KUKA KRL program: main.src, main.dat

--- main.src ---
&ACCESS RVP
&REL 135
&PARAM EDITMASK = *
&PARAM TEMPLATE = C:\KRC\Roboter\Template\vorgabe
&PARAM DISKPATH = KRC:\R1\Program
DEF main( )
;fold FRAME
DECL FRAME READY_POS
DECL FRAME stack_POS
DECL FRAME up_pos
DECL FRAME stack_end
DECL FRAME rotation_pos
DECL INT X
;endfold
;FOLD INI;%{PE}
  ;FOLD BASISTECH INI
    GLOBAL INTERRUPT DECL 3 WHEN $STOPMESS==TRUE DO IR_STOPM ( )
    INTERRUPT ON 3
    BAS (#INITMOV,0 )
  ;ENDFOLD (BASISTECH INI)
  ;FOLD USER INI
    ;Make your modifications here

  ;ENDFOLD (USER INI)
;ENDFOLD (INI)
;FOLD PTP HOME  Vel= 100 % DEFAULT;%{PE}%MKUKATPBASIS,%CMOVE,%VPTP,%P 1:PTP, 2:HOME, 3:, 5:100, 7:DEFAULT
$BWDSTART = FALSE
PDAT_ACT=PDEFAULT
FDAT_ACT=FHOME
BAS (#PTP_PARAMS,100 )
$H_POS=XHOME
PTP  XHOME
;ENDFOLD
if false then
;FOLD PTP maduo Vel=100 % PDAT1 Tool[1]:test Base[1]:tesy;%{PE}%R 8.3.44,%MKUKATPBASIS,%CMOVE,%VPTP,%P 1:PTP, 2:maduo, 3:, 5:100, 7:PDAT1
$BWDSTART=FALSE
PDAT_ACT=PPDAT1
FDAT_ACT=Fmaduo
BAS(#PTP_PARAMS,100)
PTP Xmaduo
;ENDFOLD
endif
loop
continue
$advance=3
;FOLD USER INI
$out[2]=FALSE
$OUT[3]=false
$OUT[4]=false
;ENDFOLD
$advance=3
;PTP Pick_Up
;FOLD PTP pick_up CONT Vel=100 % PDAT3 Tool[1]:test Base[1]:tesy;%{PE}%R 8.3.44,%MKUKATPBASIS,%CMOVE,%VPTP,%P 1:PTP, 2:pick_up, 3:C_DIS, 5:100, 7:PDAT3
$BWDSTART=FALSE
PDAT_ACT=PPDAT3
FDAT_ACT=Fpick_up
BAS(#PTP_PARAMS,100)
PTP Xpick_up C_DIS
;ENDFOLD
continue
;wait for $in[1] and $in[2] AND $aut ;wait allow Pick
wait sec 0
$ov_pro=100
$advance=3
;PTP pick_Up
$out[3]=true
calculation()
CONTINUE
;start rotation
;START TO MADUO
;START
;fold READY_POS
READY_POS=Xmaduo
ready_POS.X=ready_pos.X+P_POSITION[num,tier].X
ready_pos.y=ready_pos.y+P_POSITION[num,tier].y
READY_POS.Z=READY_POS.Z+RH
$BASE=BASE_DATA[1]
FOR X=1 TO 6
$VEL_AXIS[X]=85
$ACC_AXIS[X]=85
ENDFOR
$APO.CPTP=5
ptp READY_POS C_DIS
;endfold
; stack start
;FOLD STACK_POS
stack_POS=Xmaduo
stack_POS.X=stack_POS.X+P_POSITION[num,tier].X
stack_POS.y=stack_POS.y+P_POSITION[num,tier].y
$BASE=BASE_DATA[1]
FOR X=1 TO 6
$VEL_AXIS[X]=85
$ACC_AXIS[X]=85
ENDFOR
$APO.CPTP=5
ptp stack_POS C_DIS
;ENDFOLD
$OUT[2]=FALSE
$OUT[4]=true
wait sec 1
;fold READY_POS
READY_POS=Xmaduo
ready_pos.X=ready_pos.X+P_POSITION[num,tier].X
ready_pos.y=ready_pos.y+P_POSITION[num,tier].y
READY_POS.Z=READY_POS.Z+RH
$BASE=BASE_DATA[1]
FOR X=1 TO 6
$VEL_AXIS[X]=85
$ACC_AXIS[X]=85
ENDFOR
$APO.CPTP=5
ptp READY_POS C_DIS
;endfold
$advance=3
;STACK END
$out[3]=false
$out[4]=false
$ov_pro=100
;FOLD COUNT
Tier=Tier+1
if Tier>3 then
   NUM=Num+1
tier=1

endif
if num>4 then
num=1
exit
endif

;ENDFOLD
endloop
;FOLD PTP HOME Vel=100 % DEFAULT;%{PE}%R 8.3.44,%MKUKATPBASIS,%CMOVE,%VPTP,%P 1:PTP, 2:HOME, 3:, 5:100, 7:DEFAULT
$BWDSTART=FALSE
PDAT_ACT=PDEFAULT
FDAT_ACT=FHOME
BAS(#PTP_PARAMS,100)
$H_POS=XHOME
PTP XHOME
;ENDFOLD
END

--- main.dat ---
&ACCESS RVP
&REL 135
&PARAM EDITMASK = *
&PARAM TEMPLATE = C:\KRC\Roboter\Template\vorgabe
&PARAM DISKPATH = KRC:\R1\Program
DEFDAT  main
;FOLD EXTERNAL DECLARATIONS;%{PE}%MKUKATPBASIS,%CEXT,%VCOMMON,%P
;FOLD BASISTECH EXT;%{PE}%MKUKATPBASIS,%CEXT,%VEXT,%P
EXT  BAS (BAS_COMMAND  :IN,REAL  :IN )
DECL INT SUCCESS
;ENDFOLD (BASISTECH EXT)
;FOLD USER EXT;%{E}%MKUKATPUSER,%CEXT,%VEXT,%P
;Make your modifications here

;ENDFOLD (USER EXT)
;ENDFOLD (EXTERNAL DECLARATIONS)
DECL BASIS_SUGG_T LAST_BASIS={POINT1[] "frist2                  ",POINT2[] "frist2                  ",CP_PARAMS[] "CPDAT0                  ",PTP_PARAMS[] "PDAT10                  ",CONT[] "                        ",CP_VEL[] "2.0                     ",PTP_VEL[] "100                     ",SYNC_PARAMS[] "SYNCDAT                 ",SPL_NAME[] "S0                      ",A_PARAMS[] "ADAT0                   "}
DECL E6POS XMADUO={X 62.2935791,Y 139.037537,Z -69.1296539,A 92.7829361,B -2.23925900,C 179.824402,S 2,T 2,E1 0.0,E2 0.0,E3 0.0,E4 0.0,E5 0.0,E6 0.0}
DECL FDAT Fmaduo={TOOL_NO 1,BASE_NO 1,IPO_FRAME #BASE,POINT2[] " ",TQ_STATE FALSE}
DECL PDAT PPDAT1={VEL 100.000,ACC 100.000,APO_DIST 100.000,GEAR_JERK 50.0000,EXAX_IGN 0}
DECL E6POS XPICK={X -102.774834,Y 251.292023,Z 361.431549,A 101.678474,B -3.80238652,C -178.452682,S 2,T 2,E1 0.0,E2 0.0,E3 0.0,E4 0.0,E5 0.0,E6 0.0}
DECL FDAT Fpick={TOOL_NO 1,BASE_NO 1,IPO_FRAME #BASE,POINT2[] " ",TQ_STATE FALSE}
DECL PDAT PPDAT2={VEL 100.000,ACC 100.000,APO_DIST 100.000,GEAR_JERK 50.0000}
DECL E6POS XPICK_UP={X 62.2935791,Y 139.037537,Z 32.6462364,A 92.7829361,B -2.23925900,C 179.824402,S 2,T 2,E1 0.0,E2 0.0,E3 0.0,E4 0.0,E5 0.0,E6 0.0}
DECL FDAT Fpick_up={TOOL_NO 1,BASE_NO 1,IPO_FRAME #BASE,POINT2[] " ",TQ_STATE FALSE}
DECL PDAT PPDAT3={VEL 100.000,ACC 100.000,APO_DIST 100.000,APO_MODE #CDIS,GEAR_JERK 50.0000,EXAX_IGN 0}
DECL PDAT PPDAT4={VEL 100.000,ACC 100.000,APO_DIST 100.000,APO_MODE #CDIS,GEAR_JERK 50.0000}
DECL E6POS XFRIST={X 422.535797,Y -36.3018227,Z 305.408325,A -177.317154,B -2.17969489,C -178.043152,S 2,T 2,E1 0.0,E2 0.0,E3 0.0,E4 0.0,E5 0.0,E6 0.0}
DECL FDAT Ffrist={TOOL_NO 1,BASE_NO 0,IPO_FRAME #BASE,POINT2[] " ",TQ_STATE FALSE}
DECL PDAT PPDAT5={VEL 100.000,ACC 100.000,APO_DIST 100.000,GEAR_JERK 50.0000}
DECL PDAT PPDAT6={VEL 100.000,ACC 100.000,APO_DIST 100.000,GEAR_JERK 50.0000,EXAX_IGN 0}
DECL E6POS XFRIST1={X 4932.72314,Y 239.200607,Z 876.474487,A 120.238602,B 0.000230552105,C 180.000,S 2,T 43,E1 0.0,E2 0.0,E3 0.0,E4 0.0,E5 0.0,E6 0.0}
DECL FDAT Ffrist1={TOOL_NO 1,BASE_NO 1,IPO_FRAME #BASE,POINT2[] " ",TQ_STATE FALSE}
DECL PDAT PPDAT7={VEL 100.000,ACC 100.000,APO_DIST 100.000,GEAR_JERK 50.0000}
DECL E6POS XFRIST2={X 3538.39600,Y 2042.02905,Z 1538.35803,A -133.566101,B -0.000567811716,C -179.999802,S 2,T 11,E1 0.0,E2 0.0,E3 0.0,E4 0.0,E5 0.0,E6 0.0}
DECL FDAT Ffrist2={TOOL_NO 1,BASE_NO 1,IPO_FRAME #BASE,POINT2[] " ",TQ_STATE FALSE}
DECL PDAT PPDAT8={VEL 100.000,ACC 100.000,APO_DIST 100.000,GEAR_JERK 50.0000}
DECL E6POS Xrotation={X 3345.06812,Y 2038.01,Z 1538.40698,A -133.580795,B -0.000434641697,C -179.999603,S 2,T 11,E1 0.0,E2 0.0,E3 0.0,E4 0.0,E5 0.0,E6 0.0}
DECL FDAT Frotation={TOOL_NO 1,BASE_NO 1,IPO_FRAME #BASE,POINT2[] " ",TQ_STATE FALSE}
DECL PDAT PPDAT9={VEL 100.000,ACC 100.000,APO_DIST 100.000,GEAR_JERK 50.0000}
DECL PDAT PPDAT10={VEL 100.000,ACC 100.000,APO_DIST 100.000,GEAR_JERK 50.0000}
ENDDAT
